TYPE ST_GC_ServiceParam :
STRUCT
	SpinAxisJogCW : ST_GCSpinAxisJogParam;
	SpinAxisMoveAbs : ST_GCSpinAxisMoveAbsParam;
	SpinAxisMoveVelCW : ST_GCSpinAxisMoveVelParam;
	LiftPinAxisMoveVelCW : ST_GCLiftPinAxisMoveVelParam;
	LiftPinAxisMoveVelCCW : ST_GCLiftPinAxisMoveVelParam;
	LiftPinAxisMoveAbs : ST_GCLiftPinAxisMoveAbsParam;
	SingleProcess : ST_GCSingleProcessParam;
END_STRUCT
END_TYPE

(* stored: Version 1.1.0.1, ProductVersion 3.1.4026.18
   DUT ST_GC_ServiceParam: Id {9d771c70-165f-48ed-a888-a145a70861d4} *)
